TYPE ST_CtrlInPbStraightTransport :
STRUCT
	HoldExtendedRun	: BOOL;		//When set the extended run is not executed until variable is set to false. Note that Extended run has to be Activated by configuration.
END_STRUCT
END_TYPE

(* stored: Version 1.1.0.1, ProductVersion 3.1.4024.9
   DUT ST_CtrlInPbStraightTransport: Id {0a63bb4b-6c7c-4c07-9366-224239dfcfb0} *)
